(* CODESYS project PiPlate_RELAY.library
   Company: Lennart
   Version: 1.2.0.0
   DefaultNamespace: PiPlate_RELAY
   Placeholder: PlaceholderTemplate
   Author: Lennart Albertsen
   Description: Library containing device support of PiPlate RELAY Digital
   Title: PiPlate_RELAY

Project tree, tasks and I/O mapping:
  libraries: CAA Types Extern, * (CAA Technical Workgroup); Standard, * (System); SysTypes Interfaces, * (System); IoStandard, * (System); Raspberry Pi Peripherals, * (3S - Smart Software Solutions GmbH)
  global variables GCL_PiPlate_RELAY
  00000000-0000-0000-0000-000000000000|D:\CoDeSys\LibrariesV3\trunk\Intern\CAA\CAA Template\3.4.0.0 draft\Placeholder.xml
  00000000-0000-0000-0000-000000000000|D:\CoDeSys\LibrariesV3\trunk\Intern\CAA\CAA Template\3.2.0.3 draft\Prefix.pdf
  00000000-0000-0000-0000-000000000000|D:\CoDeSys\LibrariesV3\trunk\Intern\CAA\CAA Template\3.5.2.0 draft\Placeholder.xml
  function block PiPlate_RELAY [ST]: Initialize, BeforeWriteOutputs, AfterReadInputs, read8, write8
*)

// GCL_PiPlate_RELAY
VAR_GLOBAL CONSTANT
	//OUTPUT_PORT: USINT := 16#0D;
	//INPUT_PORT: USINT := 16#19;
	//IOCON: USINT := 0;
	//GPIOA: USINT := 16#14;
	//GPIOB: USINT := 16#13;
	//GPPUB: USINT := 16#0D;
	//IODIRA: USINT := 16#00;
	//IODIRB: USINT := 16#01;
DELAY_SETTLE_NS : UDINT := 40000; // 40us
DELAY_SETTLE_NSX : UDINT := 400000; // 400us
END_VAR

// PiPlate_RELAY
FUNCTION_BLOCK PiPlate_RELAY EXTENDS spi
VAR_INPUT
	RO1:BOOL; //Relay Output 1
	RO2:BOOL; //Relay Output 2
	RO3:BOOL; //Relay Output 3
	RO4:BOOL; //Relay Output 4
	RO5:BOOL; //Relay Output 5
	RO6:BOOL; //Relay Output 6
	RO7:BOOL; //Relay Output 7
END_VAR
VAR_OUTPUT
	OPR:BOOL; //Operational
END_VAR
VAR
	_byHardwareAddress: BYTE;
	BoardBaseAddress:BYTE :=24;
	BoardType:ARRAY [0..20] OF BYTE :=[0,0,0,0,80,105,45,80,108,97,116,101,32,82,69,76,65,89,0,0,0]; (*Pi-Plate RELAY*)
	digitalOut:BYTE;
	byInDO: BYTE;
	vState:INT;
	IOStatusOK:BOOL := TRUE;
	vRecArray:ARRAY [0..20] OF BYTE;
END_VAR
VAR_TEMP
	i, k: INT;
END_VAR

SUPER^();

CASE _iState OF
	0:	IF SUPER^.init() THEN
			read8(_byHardwareAddress,00,0,0,1);
			IF vRecArray[4] = _byHardwareAddress + BoardBaseAddress THEN
				read8(_byHardwareAddress,01,0,0,1);
				IF vRecArray[4] = BoardType[4] AND vRecArray[5] = BoardType[5] AND vRecArray[6] = BoardType[6] AND vRecArray[7] = BoardType[7] AND vRecArray[8] = BoardType[8] AND vRecArray[9] = BoardType[9] AND vRecArray[10] = BoardType[10] AND vRecArray[11] = BoardType[11] AND vRecArray[12] = BoardType[12] AND vRecArray[13] = BoardType[13] AND vRecArray[14] = BoardType[14] AND vRecArray[15] = BoardType[15] AND vRecArray[16] = BoardType[16] AND vRecArray[17] = BoardType[17] THEN
					_iState := 1;
				END_IF
			END_IF;
	  	END_IF
1:	_iState := 10;
10: IF _pConnector^.dwFlags = 242 OR NOT IOStatusOK THEN
		_iState:=1000;
	END_IF
1000: _iState:=0;
END_CASE
OPR := Operational AND _iState = 10;

METHOD Initialize : UDINT
VAR_INPUT
	wModuleType : UINT;
	dwInstance : UDINT;
	pConnector : POINTER TO IoConfigConnector;
END_VAR
VAR
	pParam: POINTER TO IoConfigParameter;		
	udiResult: UDINT;
END_VAR
SUPER^.Initialize(wModuleType, dwInstance, pConnector);

pParam := ConfigGetParameter(_pConnector, 1);
IF pParam <> 0 THEN
	_byHardwareAddress := IoStandard.ConfigGetParameterValueByte(pParam, ADR(udiResult));
END_IF

(*
IF _iState = 0 THEN
write8(_byHardwareAddress,15,0,0,0);
END_IF
*)
END_METHOD

METHOD BeforeWriteOutputs : INT
VAR
	i: INT;
END_VAR
SUPER^.BeforeWriteOutputs();

IF _iState = 10 THEN
		CASE vState OF
			
			0: 	//Digital Output encode
				digitalOut.0 := RO1;
				digitalOut.1 := RO2;	
				digitalOut.2 := RO3;
				digitalOut.3 := RO4;
				digitalOut.4 := RO5;
				digitalOut.5 := RO6;
				digitalOut.6 := RO7;
				write8(_byHardwareAddress,19,digitalout,0,0); //Write Digital Outputs
				vState := 1;
		
			1:	read8(_byHardwareAddress,20,0,0,1); // Get Digital Output status
				byInDO := vRecArray[4]; //DO's status feedback
				IOStatusOK := byInDO = digitalout;
				vState := 0;
		END_CASE
END_IF
END_METHOD

METHOD AfterReadInputs : INT
VAR
	//aby: ARRAY[0..13] OF BYTE;	

END_VAR
SUPER^.AfterReadInputs();
END_METHOD

// This method is used to read the data byte of one port using the following protocol:
// Byte0: hardware address + 24
// Byte1: Command
// Byte2: Parameter1
// Byte3: Parameter2
// Bytes to return are written to vRecArray
METHOD read8 : BYTE
VAR_INPUT
	byHardwareAddress: BYTE (0..7); (* hardware address *)
	CMD : BYTE;
	PARAM1 : BYTE;
	PARAM2 : BYTE;
	Bytes2return:BYTE;
END_VAR
VAR
	abyTxBuffer: ARRAY [0..3] OF BYTE;
	abyRxBuffer: ARRAY [0..20] OF BYTE;
	i:INT;
	vNothing:BOOL;
END_VAR
abyTxBuffer[0] := byHardwareAddress +24; //SPI_WRITE_CMD;
abyTxBuffer[1] := CMD;
abyTxBuffer[2] := PARAM1;
abyTxBuffer[3] := PARAM2;


IF bytes2return > 0 THEN
	IF transferExt(pabyTxBuffer:=ADR(abyTxBuffer) , pabyRxBuffer:=ADR(abyRxBuffer) , udiSpeedHz:=50000 , udiLen:=20 , uiDelayus:=5) THEN
		vRecArray := abyRxBuffer;
	ELSE
	_iState := 1000;	
	END_IF 
END_IF
END_METHOD

// This method is used to write a data byte into a port using the following protocol:
// Byte0: hardware address + 24
// Byte1: Command
// Byte2: Parameter1
// Byte3: Parameter2
// Bytes to return (not used here)
METHOD write8 : BOOL
VAR_INPUT
	byHardwareAddress: BYTE (0..7); (* hardware address *)
	CMD : BYTE;
	PARAM1 : BYTE;
	PARAM2 : BYTE;
	Bytes2return:BYTE;
	
END_VAR
VAR_OUTPUT
	
END_VAR
VAR
	abyTxBuffer: ARRAY [0..3] OF BYTE;
	abyRxTBuffer: ARRAY [0..20] OF BYTE;
	i:INT;
	y:DWORD;
END_VAR
abyTxBuffer[0] := byHardwareAddress +24; //SPI_WRITE_CMD;
abyTxBuffer[1] := CMD;
abyTxBuffer[2] := PARAM1;
abyTxBuffer[3] := PARAM2;
	
write8 := transferExt(pabyTxBuffer:=ADR(abyTxBuffer) , pabyRxBuffer:=ADR(abyRxTBuffer) , udiSpeedHz:=500000 , udiLen:=4 , uiDelayus:=1);

IF NOT write8 THEN
   _iState := 1000;
END_IF
//END_IF
END_METHOD

END_FUNCTION_BLOCK
